TYPE E_DfiRowKind :
(
	ESTOQUE_MUDANCA := 0,
	ESTOQUE_PERIODICO := 1,
	EVENTO := 2
) DINT;
END_TYPE

(* stored: Version 1.1.0.1
   DUT E_DfiRowKind: Id {d9acbff2-7af2-4937-ad29-86fb3dc611fc} *)
